TYPE FreqRegulation_Struct :
UNION
		Value : INT;
		Bits : Bits_FreqRegulation;
END_UNION
END_TYPE

(* stored: Version 1.1.0.1, ProductVersion 3.1.4022.18
   DUT FreqRegulation_Struct: Id {b28ff265-9112-40f1-9707-386f018a51b6} *)
